(* IEC 61131-3 sources: ArfBotOS/Codesys-4/ArfBotOS.fbsdev/Application.iecapp^/FUN/group/FB_GroupHandler.fb.st^/public, 4 files *)

(* ---- M_DisableGroup.meth.st ---- *)
METHOD PUBLIC M_DisableGroup : BOOL
VAR_INPUT
END_VAR

//IF NOT Error THEN
	M_DisableGroup := TRUE;
	_DisableGroup := TRUE;
//ELSE
	//M_DisableGroup := FALSE;
//END_IF
END_METHOD

(* ---- M_EnableGroup.meth.st ---- *)
METHOD PUBLIC M_EnableGroup : BOOL
VAR_INPUT
END_VAR

IF Enable AND NOT Error THEN
	M_EnableGroup := TRUE;
	_EnableGroup := TRUE;
	_GroupEnabled := FALSE;
ELSE
	M_EnableGroup := FALSE;
END_IF
END_METHOD

(* ---- M_ResetGroup.meth.st ---- *)
METHOD PUBLIC M_ResetGroup : BOOL
VAR_INPUT
END_VAR

_ResetGroup := TRUE;
END_METHOD

(* ---- M_SetKinematics.meth.st ---- *)
METHOD PUBLIC M_SetKinematics : BOOL
VAR_INPUT
	CoordinateSystem: SMC_COORD_SYSTEM;
END_VAR

IF _GroupEnabled AND NOT Error THEN
	M_SetKinematics := TRUE;
	_CoordinateSystem := CoordinateSystem;
	_SetKinematics := TRUE;
	_KinematicsSet := FALSE;
ELSE
	M_SetKinematics := FALSE;
END_IF
END_METHOD
